INTERFACE ITF_SubSystem

PROPERTY PUBLIC eCondition : SubLevelCondition
GET
END_GET
END_PROPERTY

PROPERTY PUBLIC nErrorID : UDINT
GET
END_GET
END_PROPERTY

END_INTERFACE

(* stored: Version 1.1.0.1, ProductVersion 3.1.4024.12
   Itf ITF_SubSystem: Id {6c8df39c-ed44-46e3-b018-b603526fbe5e}
   Property eCondition: Id {454336da-8f68-49f3-9a4a-bca546ed79bc}
   Get Get: Id {ac9f6269-4a59-4eab-988c-1e8ecb58cde3}
   Property nErrorID: Id {5409192a-2be2-4b7f-b274-a687c40bdb34}
   Get Get: Id {8b79048d-5120-48dd-961d-85904458209d} *)
